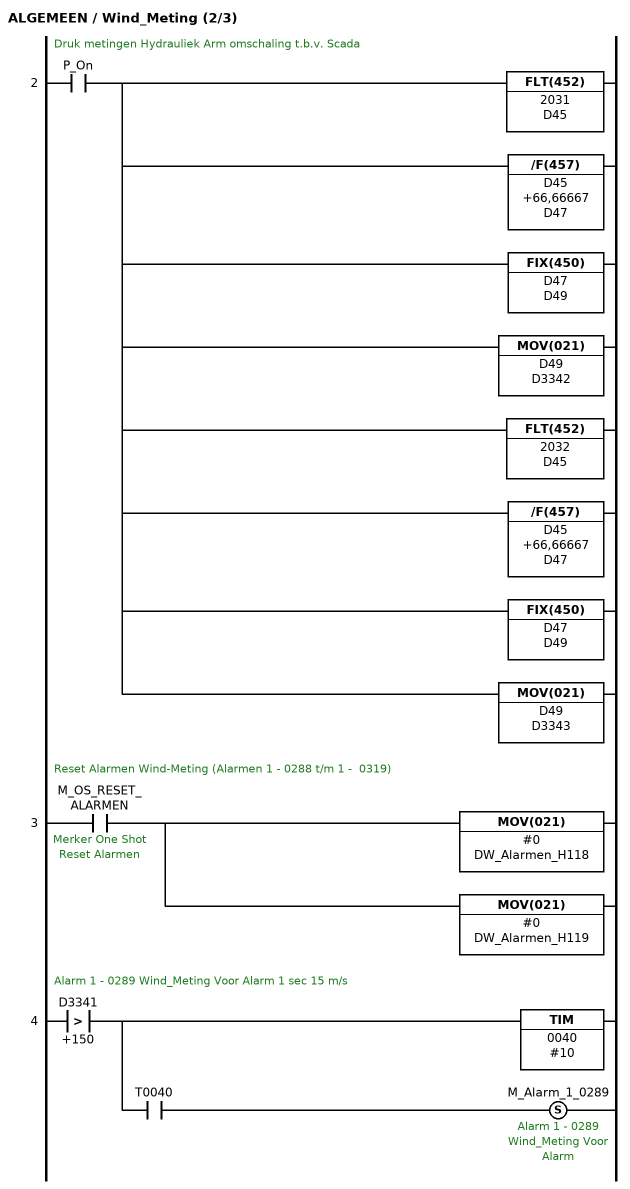
; rung 2: Druk metingen Hydrauliek Arm omschaling t.b.v. Scada
LD P_On
FLT(452) 2031 D45
/F(457) D45 +66,66667 D47
FIX(450) D47 D49
MOV(021) D49 D3342
FLT(452) 2032 D45
/F(457) D45 +66,66667 D47
FIX(450) D47 D49
MOV(021) D49 D3343
; rung 3: Reset Alarmen Wind-Meting (Alarmen 1 - 0288 t/m 1 -  0319)
LD M_OS_RESET_ALARMEN  ; Merker One Shot Reset Alarmen
MOV(021) #0 DW_Alarmen_H118
MOV(021) #0 DW_Alarmen_H119
; rung 4: Alarm 1 - 0289 Wind_Meting Voor Alarm 1 sec 15 m/s
LD>S(322) D3341 +150
TIM 0040 #10
AND T0040
SET M_Alarm_1_0289  ; Alarm 1 - 0289 Wind_Meting Voor Alarm

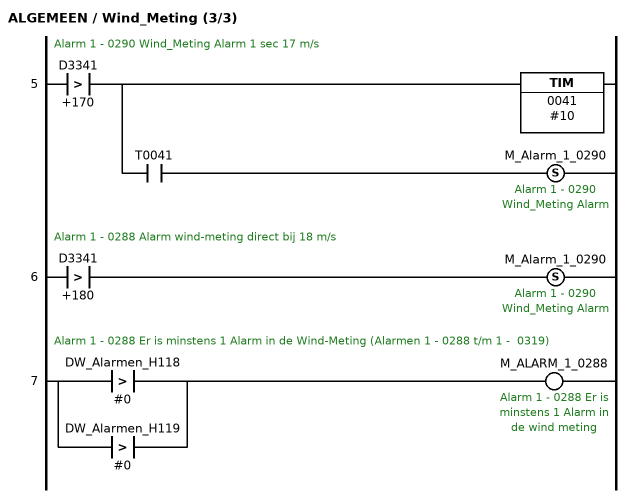
; rung 5: Alarm 1 - 0290 Wind_Meting Alarm 1 sec 17 m/s
LD>S(322) D3341 +170
TIM 0041 #10
AND T0041
SET M_Alarm_1_0290  ; Alarm 1 - 0290 Wind_Meting Alarm
; rung 6: Alarm 1 - 0288 Alarm wind-meting direct bij 18 m/s
LD>S(322) D3341 +180
SET M_Alarm_1_0290  ; Alarm 1 - 0290 Wind_Meting Alarm
; rung 7: Alarm 1 - 0288 Er is minstens 1 Alarm in de Wind-Meting (Alarmen 1 - 0288 t/m 1 -  0319)
LD>(320) DW_Alarmen_H118 #0
OR>(320) DW_Alarmen_H119 #0
OUT M_ALARM_1_0288  ; Alarm 1 - 0288 Er is minstens 1 Alarm in de wind meting

### Section Alarm_Handler

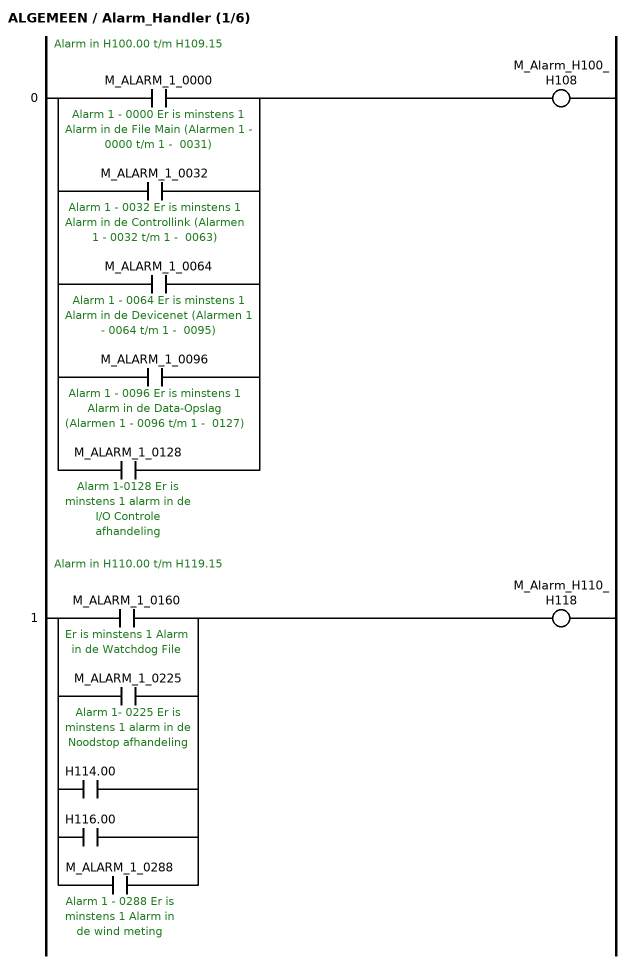
; rung 0: Alarm in H100.00 t/m H109.15
LD M_ALARM_1_0000  ; Alarm 1 - 0000 Er is minstens 1 Alarm in de File Main (Alarmen 1 - 0000 t/m 1 -  0031)
OR M_ALARM_1_0032  ; Alarm 1 - 0032 Er is minstens 1 Alarm in de Controllink (Alarmen 1 - 0032 t/m 1 -  0063)
OR M_ALARM_1_0064  ; Alarm 1 - 0064 Er is minstens 1 Alarm in de Devicenet (Alarmen 1 - 0064 t/m 1 -  0095)
OR M_ALARM_1_0096  ; Alarm 1 - 0096 Er is minstens 1 Alarm in de Data-Opslag (Alarmen 1 - 0096 t/m 1 -  0127)
OR M_ALARM_1_0128  ; Alarm 1-0128 Er is minstens 1 alarm in de I/O Controle afhandeling
OUT M_Alarm_H100_H108
; rung 1: Alarm in H110.00 t/m H119.15
LD M_ALARM_1_0160  ; Er is minstens 1 Alarm in de Watchdog File
OR M_ALARM_1_0225  ; Alarm 1- 0225 Er is minstens 1 alarm in de Noodstop afhandeling
OR H114.00
OR H116.00
OR M_ALARM_1_0288  ; Alarm 1 - 0288 Er is minstens 1 Alarm in de wind meting
OUT M_Alarm_H110_H118

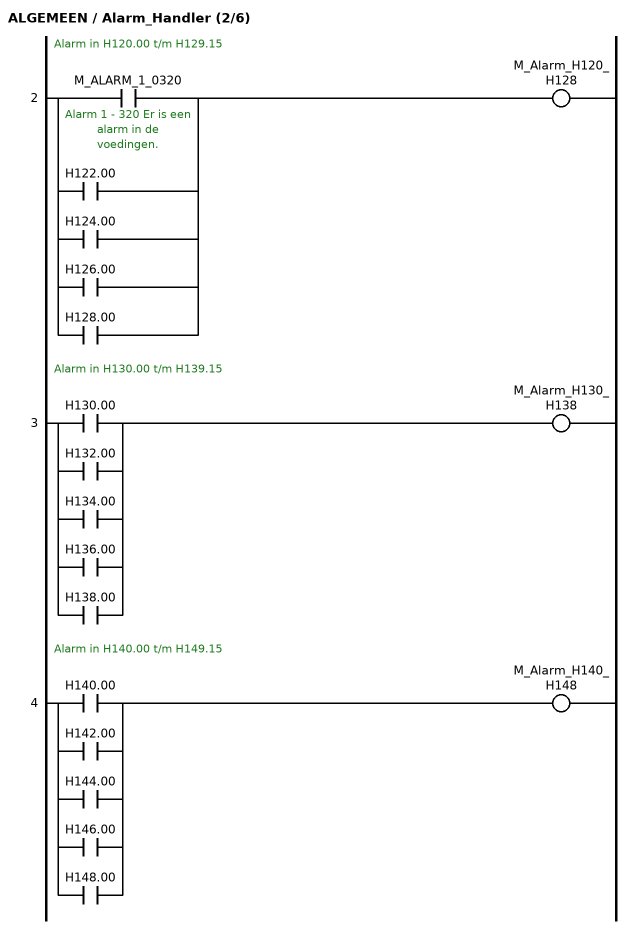
; rung 2: Alarm in H120.00 t/m H129.15
LD M_ALARM_1_0320  ; Alarm 1 - 320 Er is een alarm in de voedingen.
OR H122.00
OR H124.00
OR H126.00
OR H128.00
OUT M_Alarm_H120_H128
; rung 3: Alarm in H130.00 t/m H139.15
LD H130.00
OR H132.00
OR H134.00
OR H136.00
OR H138.00
OUT M_Alarm_H130_H138
; rung 4: Alarm in H140.00 t/m H149.15
LD H140.00
OR H142.00
OR H144.00
OR H146.00
OR H148.00
OUT M_Alarm_H140_H148

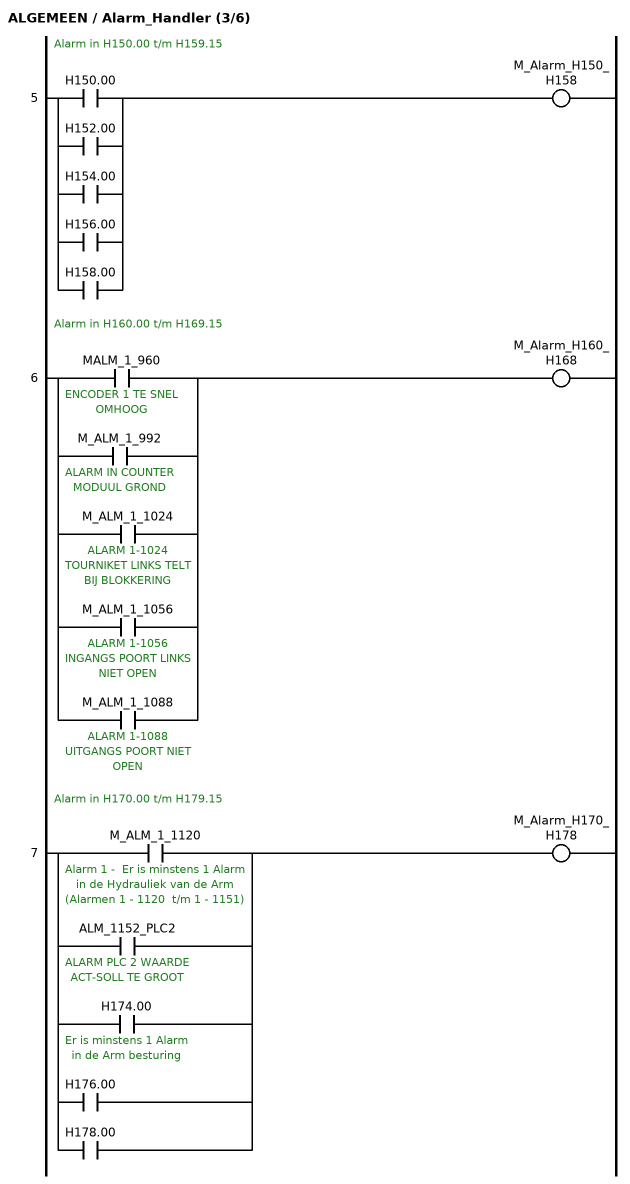
; rung 5: Alarm in H150.00 t/m H159.15
LD H150.00
OR H152.00
OR H154.00
OR H156.00
OR H158.00
OUT M_Alarm_H150_H158
; rung 6: Alarm in H160.00 t/m H169.15
LD MALM_1_960  ; ENCODER 1 TE SNEL OMHOOG
OR M_ALM_1_992  ; ALARM IN COUNTER MODUUL GROND
OR M_ALM_1_1024  ; ALARM 1-1024 TOURNIKET LINKS TELT BIJ BLOKKERING
OR M_ALM_1_1056  ; ALARM 1-1056 INGANGS POORT LINKS NIET OPEN
OR M_ALM_1_1088  ; ALARM 1-1088 UITGANGS POORT NIET OPEN
OUT M_Alarm_H160_H168
; rung 7: Alarm in H170.00 t/m H179.15
LD M_ALM_1_1120  ; Alarm 1 -  Er is minstens 1 Alarm in de Hydrauliek van de Arm  (Alarmen 1 - 1120  t/m 1 - 1151)
OR ALM_1152_PLC2  ; ALARM PLC 2 WAARDE ACT-SOLL TE GROOT
OR H174.00  ; Er is minstens 1 Alarm in de Arm besturing
OR H176.00
OR H178.00
OUT M_Alarm_H170_H178

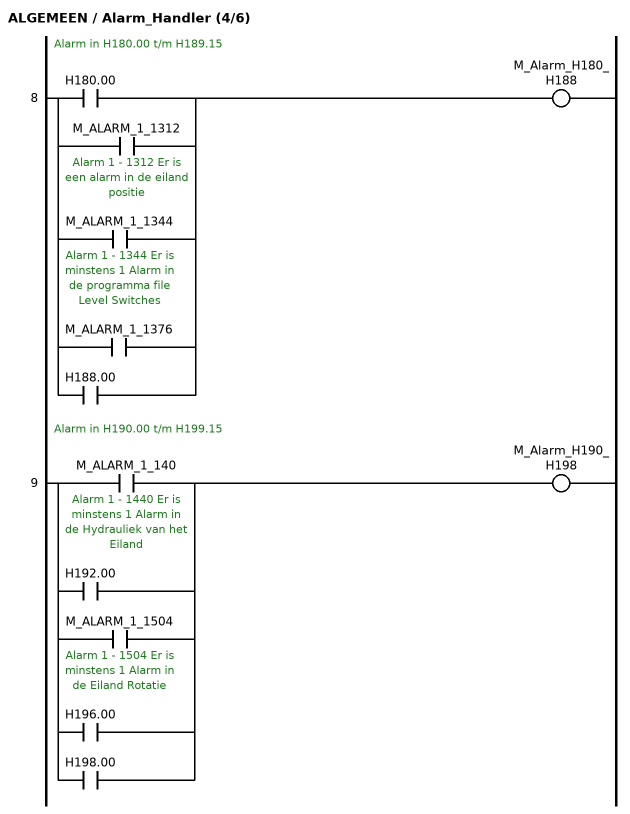
; rung 8: Alarm in H180.00 t/m H189.15
LD H180.00
OR M_ALARM_1_1312  ; Alarm 1 - 1312 Er is een alarm in de eiland positie
OR M_ALARM_1_1344  ; Alarm 1 - 1344 Er is minstens 1 Alarm in de programma file Level Switches
OR M_ALARM_1_1376
OR H188.00
OUT M_Alarm_H180_H188
; rung 9: Alarm in H190.00 t/m H199.15
LD M_ALARM_1_140  ; Alarm 1 - 1440 Er is minstens 1 Alarm in de Hydrauliek van het Eiland
OR H192.00
OR M_ALARM_1_1504  ; Alarm 1 - 1504 Er is minstens 1 Alarm in de Eiland Rotatie
OR H196.00
OR H198.00
OUT M_Alarm_H190_H198

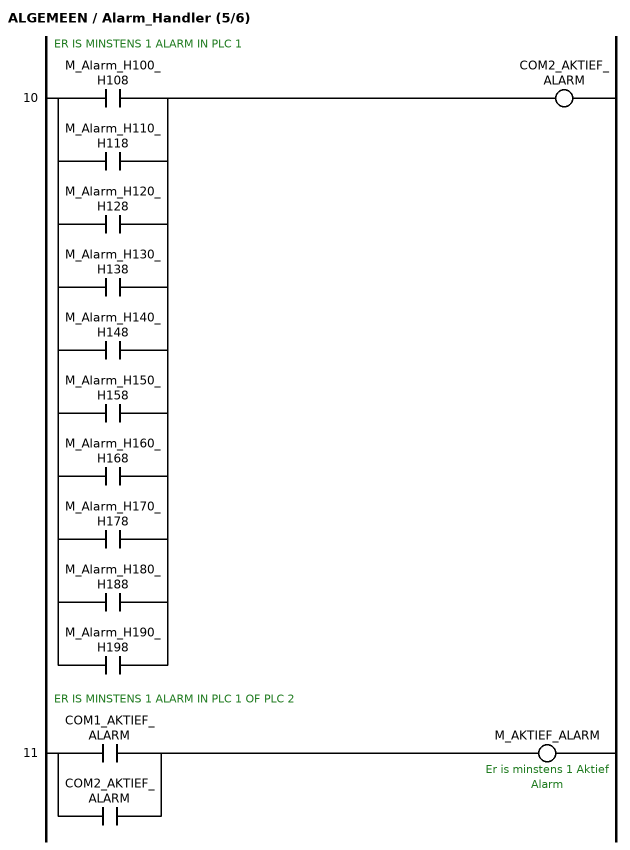
; rung 10: ER IS MINSTENS 1 ALARM IN PLC 1
LD M_Alarm_H100_H108
OR M_Alarm_H110_H118
OR M_Alarm_H120_H128
OR M_Alarm_H130_H138
OR M_Alarm_H140_H148
OR M_Alarm_H150_H158
OR M_Alarm_H160_H168
OR M_Alarm_H170_H178
OR M_Alarm_H180_H188
OR M_Alarm_H190_H198
OUT COM2_AKTIEF_ALARM
; rung 11: ER IS MINSTENS 1 ALARM IN PLC 1 OF PLC 2
LD COM1_AKTIEF_ALARM
OR COM2_AKTIEF_ALARM
OUT M_AKTIEF_ALARM  ; Er is minstens 1 Aktief Alarm

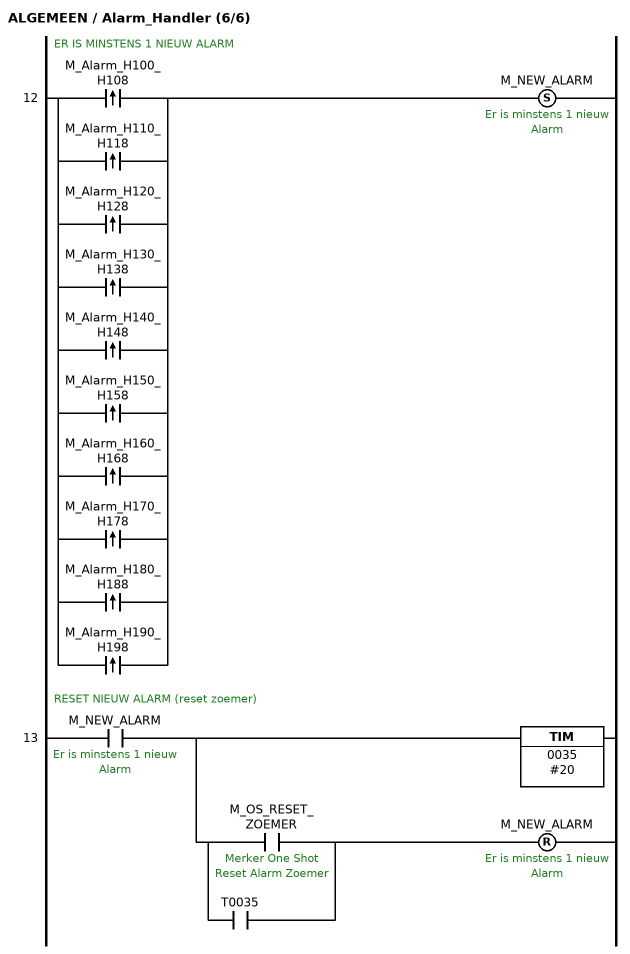
; rung 12: ER IS MINSTENS 1 NIEUW ALARM
@LD M_Alarm_H100_H108
@OR M_Alarm_H110_H118
@OR M_Alarm_H120_H128
@OR M_Alarm_H130_H138
@OR M_Alarm_H140_H148
@OR M_Alarm_H150_H158
@OR M_Alarm_H160_H168
@OR M_Alarm_H170_H178
@OR M_Alarm_H180_H188
@OR M_Alarm_H190_H198
SET M_NEW_ALARM  ; Er is minstens 1 nieuw Alarm
; rung 13: RESET NIEUW ALARM (reset zoemer)
LD M_NEW_ALARM  ; Er is minstens 1 nieuw Alarm
TIM 0035 #20
LD M_OS_RESET_ZOEMER  ; Merker One Shot Reset Alarm Zoemer
OR T0035
ANDLD
RSET M_NEW_ALARM  ; Er is minstens 1 nieuw Alarm

### Section Einde_Algemeen
; rung 0
END(001)

## Program BEDIENING_SIGNAAL (cyclic task 1)
Local symbols
Com1_44HS12 3011.15 BOOL
Com1_44HS124 3012.00 BOOL
Com1_SK_Open_Linker_Ingangs_Poortje_Eiland 3014.09 BOOL
Com1_SK_Open_Linker_Ingangs_Poortje_Oever 3014.11 BOOL
Com1_SK_Open_Linker_Uitgangs_Poortjes_Eiland 3014.13 BOOL
Com1_SK_Open_Rechter_Ingangs_Poortje_Eiland 3014.10 BOOL
Com1_SK_Open_Rechter_Ingangs_Poortje_Oever 3014.12 BOOL
Com1_SK_Open_Rechter_Uitgangs_Poortje_Eiland 3014.14 BOOL
Com1_SK_Open_Sluit_Linker_Oever_Poortjes_ 3014.05 BOOL
Com1_SK_Open_Sluit_Rechter_Oever_Poortjes_ 3014.06 BOOL
Com1_SK_Open_Uitgangs_Poortjes_Oever 3014.15 BOOL
Com1_SK_Reset_Alarmen 3014.01 BOOL
Com1_SK_SPARE_3314_00 3014.00 BOOL
Com1_SK_SPARE_3314_02 3014.02 BOOL
Com1_SK_SPARE_3315_03 3015.02 BOOL
Com1_SK_SPARE_3315_07 3015.07 BOOL
Com1_SK_SPARE_3315_08 3015.08 BOOL
Com1_SK_SPARE_3315_09 3015.09 BOOL
Com1_SK_Stabilisatie_Eiland_Linksom 3015.05 BOOL
Com1_SK_Stabilisatie_Eiland_Rechtsom 3015.06 BOOL
Com1_SK_Start_Stop_Hoofdpomp_Arm 3015.01 BOOL
Com1_SK_Start_Stop_Hoofdpomp_Eiland 3015.04 BOOL
Com1_SK_Start_Stop_Hydrau 3014.03 BOOL
Com1_SK_Start_Stop_Show 3014.04 BOOL
Com1_SK_Start_Stop_Stuurpomp_Arm 3015.00 BOOL
Com1_SK_Start_Stop_Stuurpomp_Eiland 3015.03 BOOL
Com1_SK_Vrijgave_Linker_Tourniquet 3014.07 BOOL
Com1_SK_Vrijgave_Rechter_Tourniquet 3014.08 BOOL
Com1_SK_WCD_1 3015.10 BOOL
Com1_SK_WCD_2 3015.11 BOOL
Com1_SK_WCD_3 3015.12 BOOL
Com1_SK_WCD_4 3015.13 BOOL
Com1_SK_WCD_5 3015.14 BOOL
Com1_SK_WCD_6 3015.15 BOOL
Com2_44HS14 3312.00 BOOL
Com2_SK_Open_Linker_Ingangs_Poortje_Eiland 3314.09 BOOL  ; Skada Bediening Open Linker Ingangs Poortje Eiland
Com2_SK_Open_Linker_Ingangs_Poortje_Oever 3314.11 BOOL  ; Skada Bediening Open Linker Ingangs Poortje Oever
Com2_SK_Open_Linker_Uitgangs_Poortjes_Eiland 3314.13 BOOL  ; Skada Bediening Open Linker Uitgangs Poortje Eiland
Com2_SK_Open_Rechter_Ingangs_Poortje_Eiland 3314.10 BOOL  ; Skada Bediening Open Rechter ingangs poortje Eiland
Com2_SK_Open_Rechter_Ingangs_Poortje_Oever 3314.12 BOOL  ; Skada Bediening Open Rechter ingangs poortje Oever
Com2_SK_Open_Rechter_Uitgangs_Poortje_Eiland 3314.14 BOOL  ; Skada Bediening Open Rechter Uitgangs poortje Eiland
Com2_SK_Open_Sluit_Linker_Oever_Poortjes_ 3314.05 BOOL  ; Skada Bediening Open / Sluit Linker Oever Poortjes
Com2_SK_Open_Sluit_Rechter_Oever_Poortjes_ 3314.06 BOOL  ; Skada Bediening Open / Sluit Rechter Oever Poortjes
Com2_SK_Open_Uitgangs_Poortjes_Oever 3314.15 BOOL  ; Skada Bediening Open Uitgangs poortjes Oever
Com2_SK_Reset_Alarmen 3314.01 BOOL  ; Skada Bediening Reset Alarmen
Com2_SK_SPARE_3314_00 3314.00 BOOL
Com2_SK_SPARE_3314_02 3314.02 BOOL
Com2_SK_SPARE_3315_03 3315.02 BOOL
Com2_SK_SPARE_3315_07 3315.07 BOOL
Com2_SK_SPARE_3315_08 3315.08 BOOL
Com2_SK_SPARE_3315_09 3315.09 BOOL
Com2_SK_Stabilisatie_Eiland_Linksom 3315.05 BOOL  ; Skada Bediening Eiland Stabilisatie Linksom
Com2_SK_Stabilisatie_Eiland_Rechtsom 3315.06 BOOL  ; Skada Bediening Eiland Stabilisatie Rechtsom
Com2_SK_Start_Stop_Hoofdpomp_Arm 3315.01 BOOL  ; Skada Bediening Start / Stop Hydrauliek Hoofdpomp Arm
Com2_SK_Start_Stop_Hoofdpomp_Eiland 3315.04 BOOL  ; Skada Bediening Start / Stop Hydrauliek Hoofdpomp Eiland
Com2_SK_Start_Stop_Hydrau 3314.03 BOOL  ; Skada Bediening Start / Stop Hydrauliek Arm & Eiland
Com2_SK_Start_Stop_Show 3314.04 BOOL  ; Skada Bediening Start / Stop Show
Com2_SK_Start_Stop_Stuurpomp_Arm 3315.00 BOOL  ; Skada Bediening Start / Stop Hydrauliek Stuurpomp Arm
Com2_SK_Start_Stop_Stuurpomp_Eiland 3315.03 BOOL  ; Skada Bediening Start / Stop Hydrauliek Stuurpomp Eiland
Com2_SK_Vrijgave_Linker_Tourniquet 3314.07 BOOL  ; Skada bediening Vrijgave Linker Tourniquets
Com2_SK_Vrijgave_Rechter_Tourniquet 3314.08 BOOL  ; Skada Bediening Vrijgave Rechter Tourniquets
Com2_SK_WCD_1 3315.10 BOOL  ; Skada Bediening Wandcontactdoos 1
Com2_SK_WCD_2 3315.11 BOOL  ; Skada Bediening Wandcontactdoos 2
Com2_SK_WCD_3 3315.12 BOOL  ; Skada Bediening Wandcontactdoos 3
Com2_SK_WCD_4 3315.13 BOOL  ; Skada Bediening Wandcontactdoos 4
Com2_SK_WCD_5 3315.14 BOOL  ; Skada Bediening Wandcontactdoos 5
Com2_SK_WCD_6 3315.15 BOOL  ; Skada Bediening Wandcontactdoos 6
Delay_Timer_Lamp_Test 0055 NUMBER  ; Delay Timer t.b.v. de lampen test
M_Hydrauliek_x_tijd_aan W56.03 BOOL  ; Hydrauliek x tijd laten door lopen nadat mode is veranderd

### Section Bediening_Scada

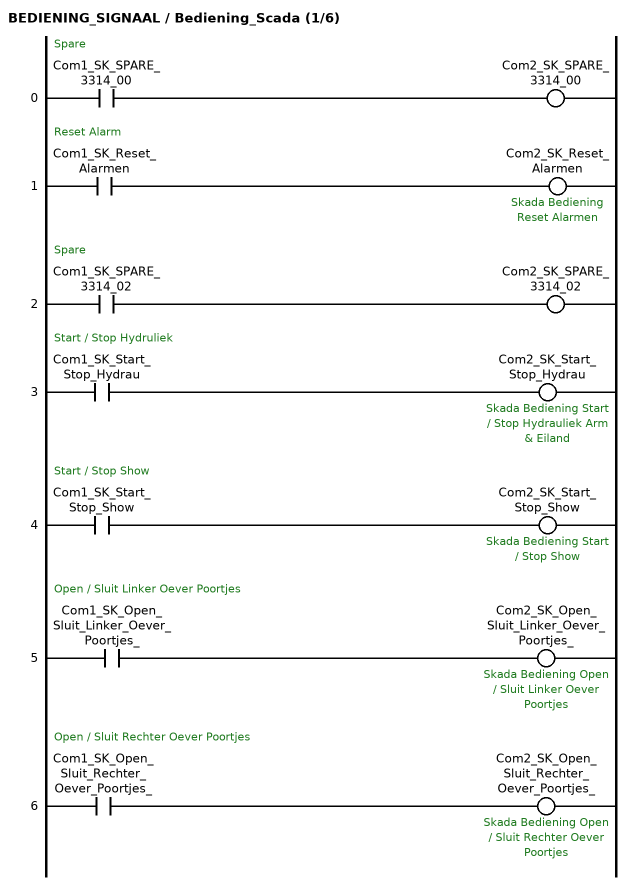
; rung 0: Spare
LD Com1_SK_SPARE_3314_00
OUT Com2_SK_SPARE_3314_00
; rung 1: Reset Alarm
LD Com1_SK_Reset_Alarmen
OUT Com2_SK_Reset_Alarmen  ; Skada Bediening Reset Alarmen
; rung 2: Spare
LD Com1_SK_SPARE_3314_02
OUT Com2_SK_SPARE_3314_02
; rung 3: Start / Stop Hydruliek
LD Com1_SK_Start_Stop_Hydrau
OUT Com2_SK_Start_Stop_Hydrau  ; Skada Bediening Start / Stop Hydrauliek Arm & Eiland
; rung 4: Start / Stop Show
LD Com1_SK_Start_Stop_Show
OUT Com2_SK_Start_Stop_Show  ; Skada Bediening Start / Stop Show
; rung 5: Open / Sluit Linker Oever Poortjes
LD Com1_SK_Open_Sluit_Linker_Oever_Poortjes_
OUT Com2_SK_Open_Sluit_Linker_Oever_Poortjes_  ; Skada Bediening Open / Sluit Linker Oever Poortjes
; rung 6: Open / Sluit Rechter Oever Poortjes
LD Com1_SK_Open_Sluit_Rechter_Oever_Poortjes_
OUT Com2_SK_Open_Sluit_Rechter_Oever_Poortjes_  ; Skada Bediening Open / Sluit Rechter Oever Poortjes

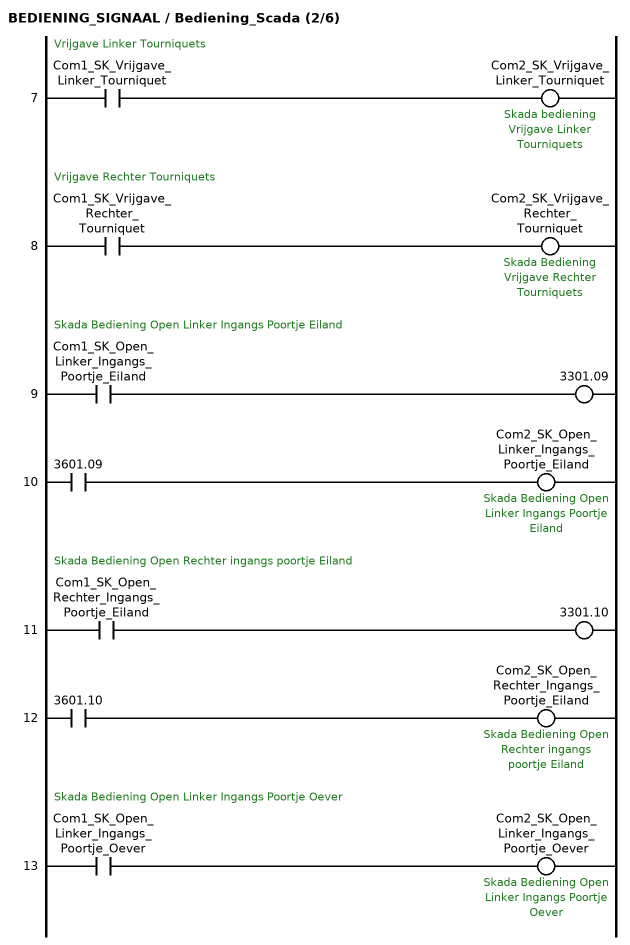
; rung 7: Vrijgave Linker Tourniquets
LD Com1_SK_Vrijgave_Linker_Tourniquet
OUT Com2_SK_Vrijgave_Linker_Tourniquet  ; Skada bediening Vrijgave Linker Tourniquets
; rung 8: Vrijgave Rechter Tourniquets
LD Com1_SK_Vrijgave_Rechter_Tourniquet
OUT Com2_SK_Vrijgave_Rechter_Tourniquet  ; Skada Bediening Vrijgave Rechter Tourniquets
; rung 9: Skada Bediening Open Linker Ingangs Poortje Eiland
LD Com1_SK_Open_Linker_Ingangs_Poortje_Eiland
OUT 3301.09
; rung 10
LD 3601.09
OUT Com2_SK_Open_Linker_Ingangs_Poortje_Eiland  ; Skada Bediening Open Linker Ingangs Poortje Eiland
; rung 11: Skada Bediening Open Rechter ingangs poortje Eiland
LD Com1_SK_Open_Rechter_Ingangs_Poortje_Eiland
OUT 3301.10
; rung 12
LD 3601.10
OUT Com2_SK_Open_Rechter_Ingangs_Poortje_Eiland  ; Skada Bediening Open Rechter ingangs poortje Eiland
; rung 13: Skada Bediening Open Linker Ingangs Poortje Oever
LD Com1_SK_Open_Linker_Ingangs_Poortje_Oever
OUT Com2_SK_Open_Linker_Ingangs_Poortje_Oever  ; Skada Bediening Open Linker Ingangs Poortje Oever

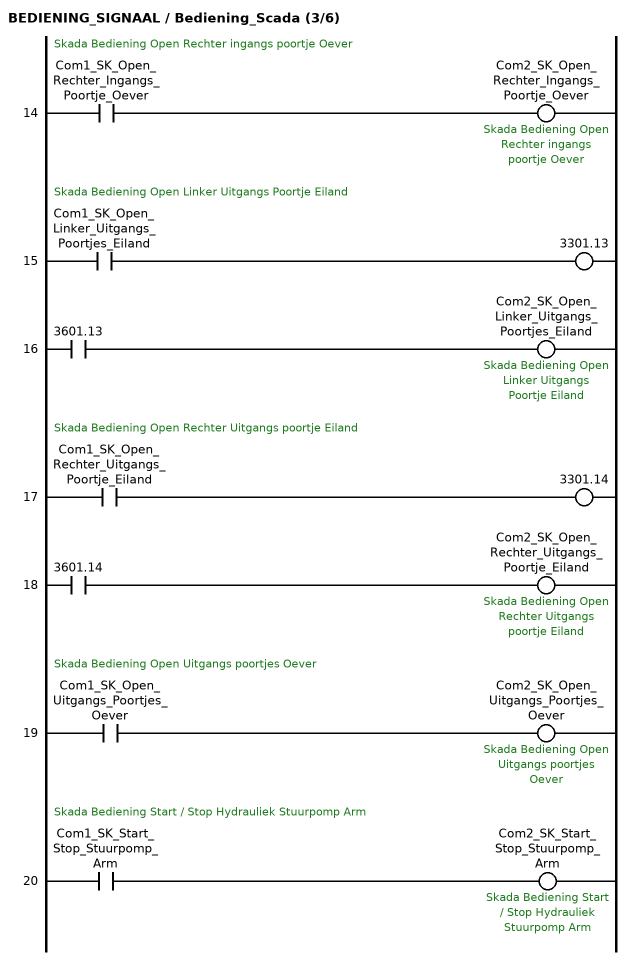
; rung 14: Skada Bediening Open Rechter ingangs poortje Oever
LD Com1_SK_Open_Rechter_Ingangs_Poortje_Oever
OUT Com2_SK_Open_Rechter_Ingangs_Poortje_Oever  ; Skada Bediening Open Rechter ingangs poortje Oever
; rung 15: Skada Bediening Open Linker Uitgangs Poortje Eiland
LD Com1_SK_Open_Linker_Uitgangs_Poortjes_Eiland
OUT 3301.13
; rung 16
LD 3601.13
OUT Com2_SK_Open_Linker_Uitgangs_Poortjes_Eiland  ; Skada Bediening Open Linker Uitgangs Poortje Eiland
; rung 17: Skada Bediening Open Rechter Uitgangs poortje Eiland
LD Com1_SK_Open_Rechter_Uitgangs_Poortje_Eiland
OUT 3301.14
; rung 18
LD 3601.14
OUT Com2_SK_Open_Rechter_Uitgangs_Poortje_Eiland  ; Skada Bediening Open Rechter Uitgangs poortje Eiland
; rung 19: Skada Bediening Open Uitgangs poortjes Oever
LD Com1_SK_Open_Uitgangs_Poortjes_Oever
OUT Com2_SK_Open_Uitgangs_Poortjes_Oever  ; Skada Bediening Open Uitgangs poortjes Oever
; rung 20: Skada Bediening Start / Stop Hydrauliek Stuurpomp Arm
LD Com1_SK_Start_Stop_Stuurpomp_Arm
OUT Com2_SK_Start_Stop_Stuurpomp_Arm  ; Skada Bediening Start / Stop Hydrauliek Stuurpomp Arm

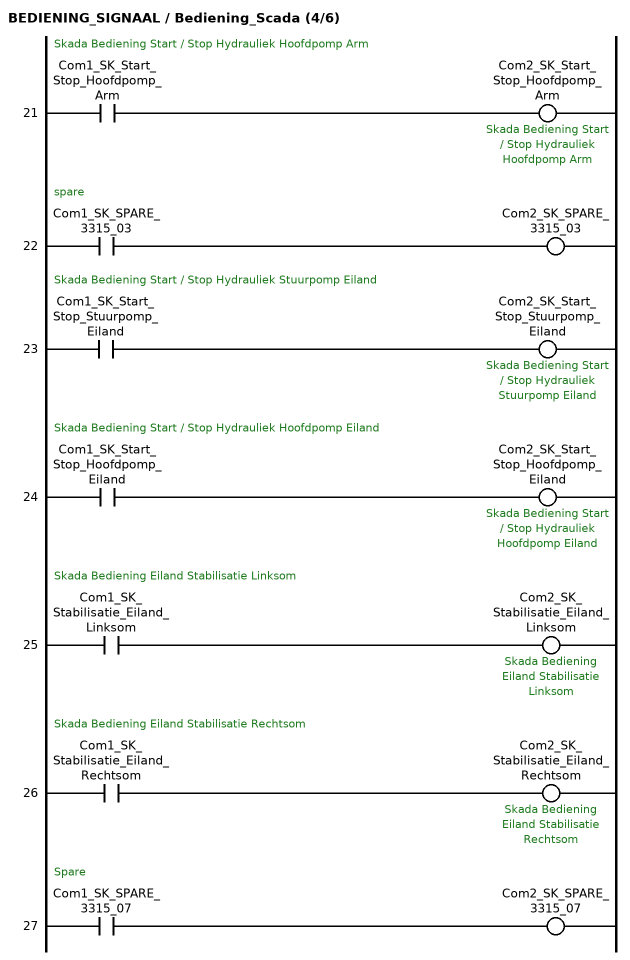
; rung 21: Skada Bediening Start / Stop Hydrauliek Hoofdpomp Arm
LD Com1_SK_Start_Stop_Hoofdpomp_Arm
OUT Com2_SK_Start_Stop_Hoofdpomp_Arm  ; Skada Bediening Start / Stop Hydrauliek Hoofdpomp Arm
; rung 22: spare
LD Com1_SK_SPARE_3315_03
OUT Com2_SK_SPARE_3315_03
; rung 23: Skada Bediening Start / Stop Hydrauliek Stuurpomp Eiland
LD Com1_SK_Start_Stop_Stuurpomp_Eiland
OUT Com2_SK_Start_Stop_Stuurpomp_Eiland  ; Skada Bediening Start / Stop Hydrauliek Stuurpomp Eiland
; rung 24: Skada Bediening Start / Stop Hydrauliek Hoofdpomp Eiland
LD Com1_SK_Start_Stop_Hoofdpomp_Eiland
OUT Com2_SK_Start_Stop_Hoofdpomp_Eiland  ; Skada Bediening Start / Stop Hydrauliek Hoofdpomp Eiland
; rung 25: Skada Bediening Eiland Stabilisatie Linksom
LD Com1_SK_Stabilisatie_Eiland_Linksom
OUT Com2_SK_Stabilisatie_Eiland_Linksom  ; Skada Bediening Eiland Stabilisatie Linksom
; rung 26: Skada Bediening Eiland Stabilisatie Rechtsom
LD Com1_SK_Stabilisatie_Eiland_Rechtsom
OUT Com2_SK_Stabilisatie_Eiland_Rechtsom  ; Skada Bediening Eiland Stabilisatie Rechtsom
; rung 27: Spare
LD Com1_SK_SPARE_3315_07
OUT Com2_SK_SPARE_3315_07

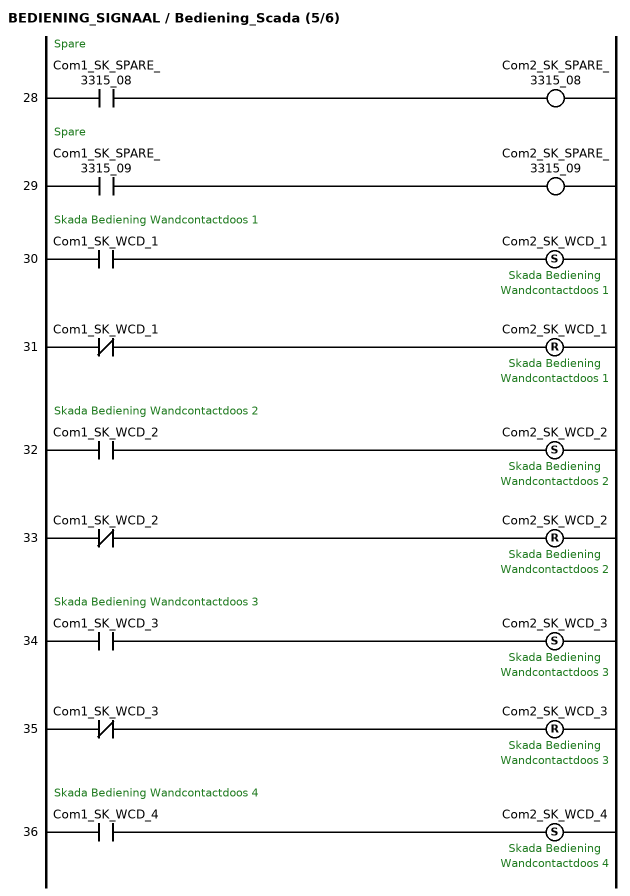
; rung 28: Spare
LD Com1_SK_SPARE_3315_08
OUT Com2_SK_SPARE_3315_08
; rung 29: Spare
LD Com1_SK_SPARE_3315_09
OUT Com2_SK_SPARE_3315_09
; rung 30: Skada Bediening Wandcontactdoos 1
LD Com1_SK_WCD_1
SET Com2_SK_WCD_1  ; Skada Bediening Wandcontactdoos 1
; rung 31
LDNOT Com1_SK_WCD_1
RSET Com2_SK_WCD_1  ; Skada Bediening Wandcontactdoos 1
; rung 32: Skada Bediening Wandcontactdoos 2
LD Com1_SK_WCD_2
SET Com2_SK_WCD_2  ; Skada Bediening Wandcontactdoos 2
; rung 33
LDNOT Com1_SK_WCD_2
RSET Com2_SK_WCD_2  ; Skada Bediening Wandcontactdoos 2
; rung 34: Skada Bediening Wandcontactdoos 3
LD Com1_SK_WCD_3
SET Com2_SK_WCD_3  ; Skada Bediening Wandcontactdoos 3
; rung 35
LDNOT Com1_SK_WCD_3
RSET Com2_SK_WCD_3  ; Skada Bediening Wandcontactdoos 3
; rung 36: Skada Bediening Wandcontactdoos 4
LD Com1_SK_WCD_4
SET Com2_SK_WCD_4  ; Skada Bediening Wandcontactdoos 4

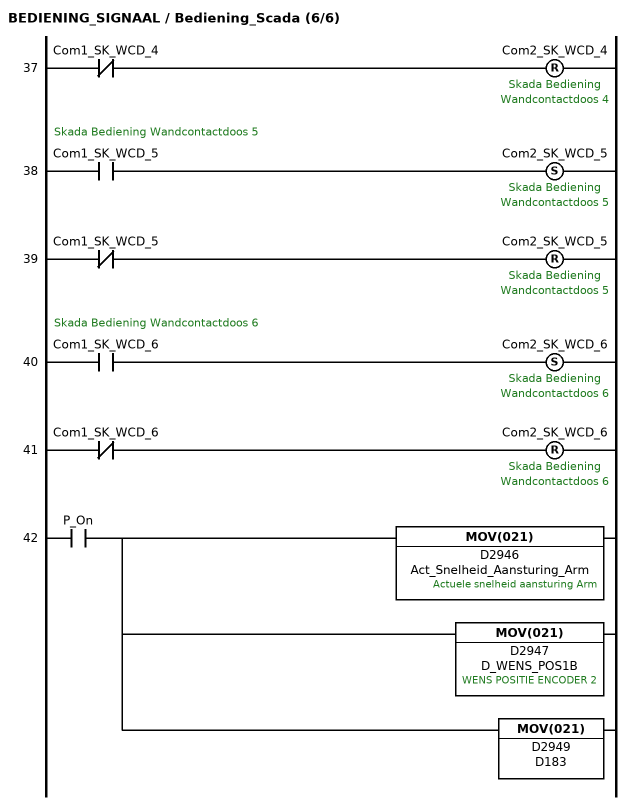
; rung 37
LDNOT Com1_SK_WCD_4
RSET Com2_SK_WCD_4  ; Skada Bediening Wandcontactdoos 4
; rung 38: Skada Bediening Wandcontactdoos 5
LD Com1_SK_WCD_5
SET Com2_SK_WCD_5  ; Skada Bediening Wandcontactdoos 5
; rung 39
LDNOT Com1_SK_WCD_5
RSET Com2_SK_WCD_5  ; Skada Bediening Wandcontactdoos 5
; rung 40: Skada Bediening Wandcontactdoos 6
LD Com1_SK_WCD_6
SET Com2_SK_WCD_6  ; Skada Bediening Wandcontactdoos 6
; rung 41
LDNOT Com1_SK_WCD_6
RSET Com2_SK_WCD_6  ; Skada Bediening Wandcontactdoos 6
; rung 42
LD P_On
MOV(021) D2946 Act_Snelheid_Aansturing_Arm  ; Actuele snelheid aansturing Arm
MOV(021) D2947 D_WENS_POS1B  ; WENS POSITIE ENCODER 2
MOV(021) D2949 D183

### Section Signalering_Scada

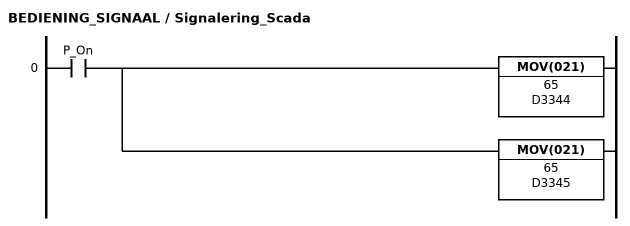
; rung 0
LD P_On
MOV(021) 65 D3344
MOV(021) 65 D3345

### Section Bediening_Grond

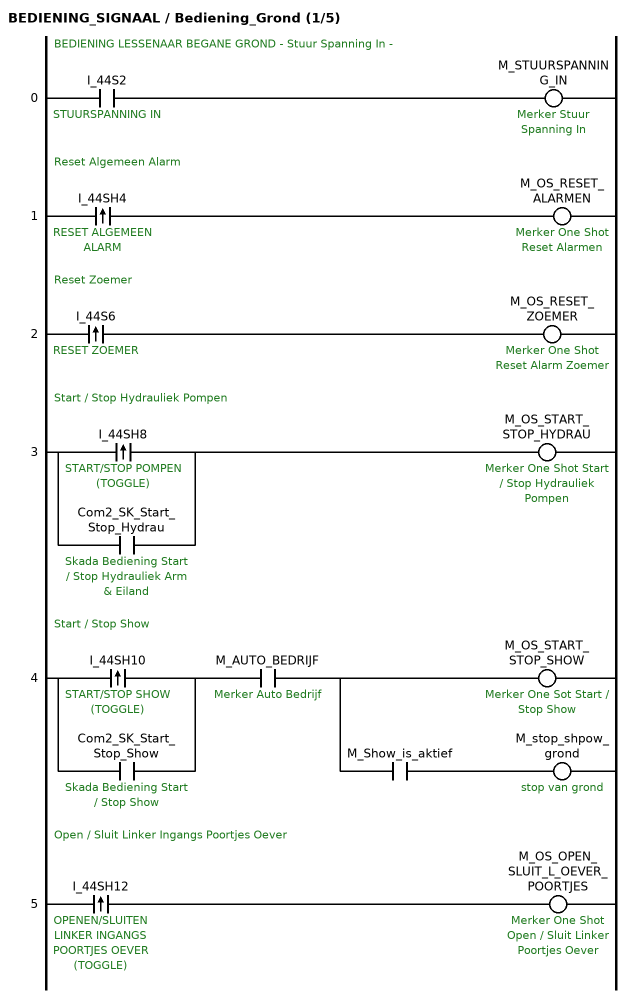
; rung 0: BEDIENING LESSENAAR BEGANE GROND - Stuur Spanning In -
LD I_44S2  ; STUURSPANNING IN
OUT M_STUURSPANNING_IN  ; Merker Stuur Spanning In
; rung 1: Reset Algemeen Alarm
@LD I_44SH4  ; RESET ALGEMEEN ALARM
OUT M_OS_RESET_ALARMEN  ; Merker One Shot Reset Alarmen
; rung 2: Reset Zoemer
@LD I_44S6  ; RESET ZOEMER
OUT M_OS_RESET_ZOEMER  ; Merker One Shot Reset Alarm Zoemer
; rung 3: Start / Stop Hydrauliek Pompen
@LD I_44SH8  ; START/STOP POMPEN (TOGGLE)
OR Com2_SK_Start_Stop_Hydrau  ; Skada Bediening Start / Stop Hydrauliek Arm & Eiland
OUT M_OS_START_STOP_HYDRAU  ; Merker One Shot Start / Stop Hydrauliek Pompen
; rung 4: Start / Stop Show
@LD I_44SH10  ; START/STOP SHOW (TOGGLE)
OR Com2_SK_Start_Stop_Show  ; Skada Bediening Start / Stop Show
AND M_AUTO_BEDRIJF  ; Merker Auto Bedrijf
OUT M_OS_START_STOP_SHOW  ; Merker One Sot Start / Stop Show
AND M_Show_is_aktief
OUT M_stop_shpow_grond  ; stop van grond
; rung 5: Open / Sluit Linker Ingangs Poortjes Oever
@LD I_44SH12  ; OPENEN/SLUITEN LINKER INGANGS POORTJES OEVER  (TOGGLE)
OUT M_OS_OPEN_SLUIT_L_OEVER_POORTJES  ; Merker One Shot Open / Sluit Linker Poortjes Oever

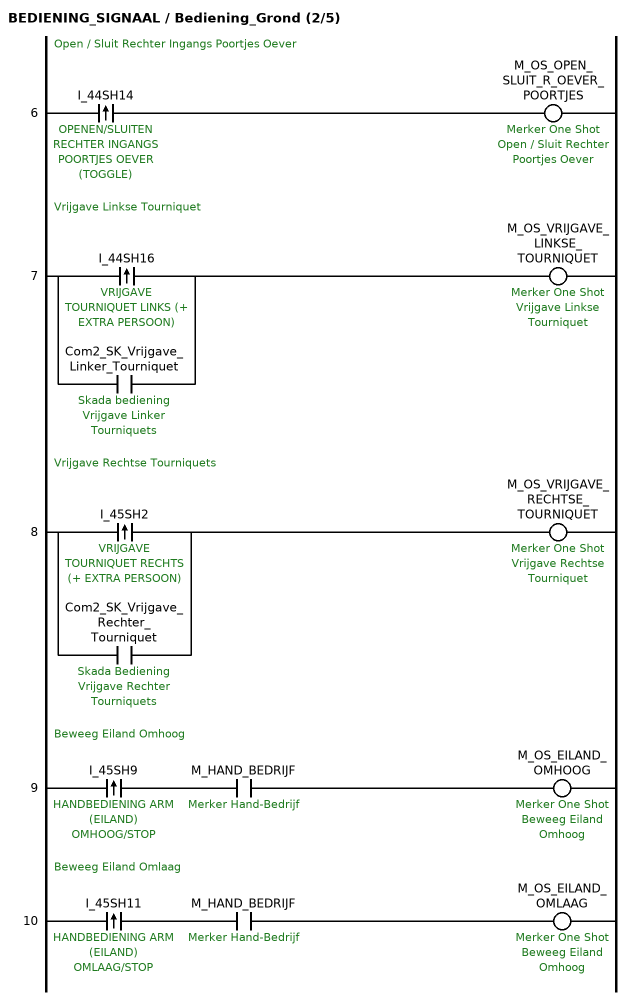
; rung 6: Open / Sluit Rechter Ingangs Poortjes Oever
@LD I_44SH14  ; OPENEN/SLUITEN RECHTER INGANGS POORTJES OEVER  (TOGGLE)
OUT M_OS_OPEN_SLUIT_R_OEVER_POORTJES  ; Merker One Shot Open / Sluit Rechter Poortjes Oever
; rung 7: Vrijgave Linkse Tourniquet
@LD I_44SH16  ; VRIJGAVE TOURNIQUET LINKS (+ EXTRA PERSOON)
OR Com2_SK_Vrijgave_Linker_Tourniquet  ; Skada bediening Vrijgave Linker Tourniquets
OUT M_OS_VRIJGAVE_LINKSE_TOURNIQUET  ; Merker One Shot Vrijgave Linkse Tourniquet
; rung 8: Vrijgave Rechtse Tourniquets
@LD I_45SH2  ; VRIJGAVE TOURNIQUET RECHTS (+ EXTRA PERSOON)
OR Com2_SK_Vrijgave_Rechter_Tourniquet  ; Skada Bediening Vrijgave Rechter Tourniquets
OUT M_OS_VRIJGAVE_RECHTSE_TOURNIQUET  ; Merker One Shot Vrijgave Rechtse Tourniquet
; rung 9: Beweeg Eiland Omhoog
@LD I_45SH9  ; HANDBEDIENING ARM (EILAND) OMHOOG/STOP
AND M_HAND_BEDRIJF  ; Merker Hand-Bedrijf
OUT M_OS_EILAND_OMHOOG  ; Merker One Shot Beweeg Eiland Omhoog
; rung 10: Beweeg Eiland Omlaag
@LD I_45SH11  ; HANDBEDIENING ARM (EILAND) OMLAAG/STOP
AND M_HAND_BEDRIJF  ; Merker Hand-Bedrijf
OUT M_OS_EILAND_OMLAAG  ; Merker One Shot Beweeg Eiland Omhoog

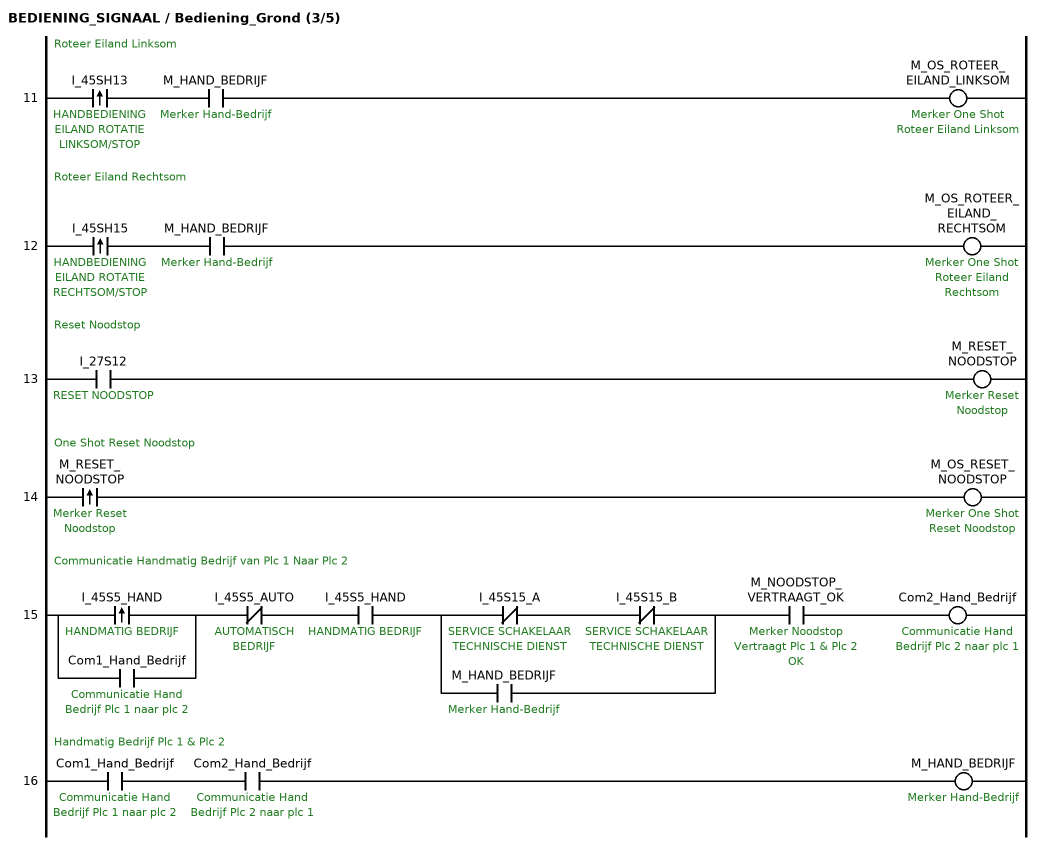
; rung 11: Roteer Eiland Linksom
@LD I_45SH13  ; HANDBEDIENING EILAND ROTATIE LINKSOM/STOP
AND M_HAND_BEDRIJF  ; Merker Hand-Bedrijf
OUT M_OS_ROTEER_EILAND_LINKSOM  ; Merker One Shot Roteer Eiland Linksom
; rung 12: Roteer Eiland Rechtsom
@LD I_45SH15  ; HANDBEDIENING EILAND ROTATIE RECHTSOM/STOP
AND M_HAND_BEDRIJF  ; Merker Hand-Bedrijf
OUT M_OS_ROTEER_EILAND_RECHTSOM  ; Merker One Shot Roteer Eiland Rechtsom
; rung 13: Reset Noodstop
LD I_27S12  ; RESET NOODSTOP
OUT M_RESET_NOODSTOP  ; Merker Reset Noodstop
; rung 14: One Shot Reset Noodstop
@LD M_RESET_NOODSTOP  ; Merker Reset Noodstop
OUT M_OS_RESET_NOODSTOP  ; Merker One Shot  Reset Noodstop
; rung 15: Communicatie Handmatig Bedrijf van Plc 1 Naar Plc 2
@LD I_45S5_HAND  ; HANDMATIG BEDRIJF
OR Com1_Hand_Bedrijf  ; Communicatie Hand Bedrijf Plc 1 naar plc 2
ANDNOT I_45S5_AUTO  ; AUTOMATISCH BEDRIJF
AND I_45S5_HAND  ; HANDMATIG BEDRIJF
LDNOT I_45S15_A  ; SERVICE SCHAKELAAR TECHNISCHE DIENST
ANDNOT I_45S15_B  ; SERVICE SCHAKELAAR TECHNISCHE DIENST
OR M_HAND_BEDRIJF  ; Merker Hand-Bedrijf
ANDLD
AND M_NOODSTOP_VERTRAAGT_OK  ; Merker Noodstop Vertraagt Plc 1 & Plc 2 OK
OUT Com2_Hand_Bedrijf  ; Communicatie Hand Bedrijf Plc 2 naar plc 1
; rung 16: Handmatig Bedrijf Plc 1 & Plc 2
LD Com1_Hand_Bedrijf  ; Communicatie Hand Bedrijf Plc 1 naar plc 2
AND Com2_Hand_Bedrijf  ; Communicatie Hand Bedrijf Plc 2 naar plc 1
OUT M_HAND_BEDRIJF  ; Merker Hand-Bedrijf

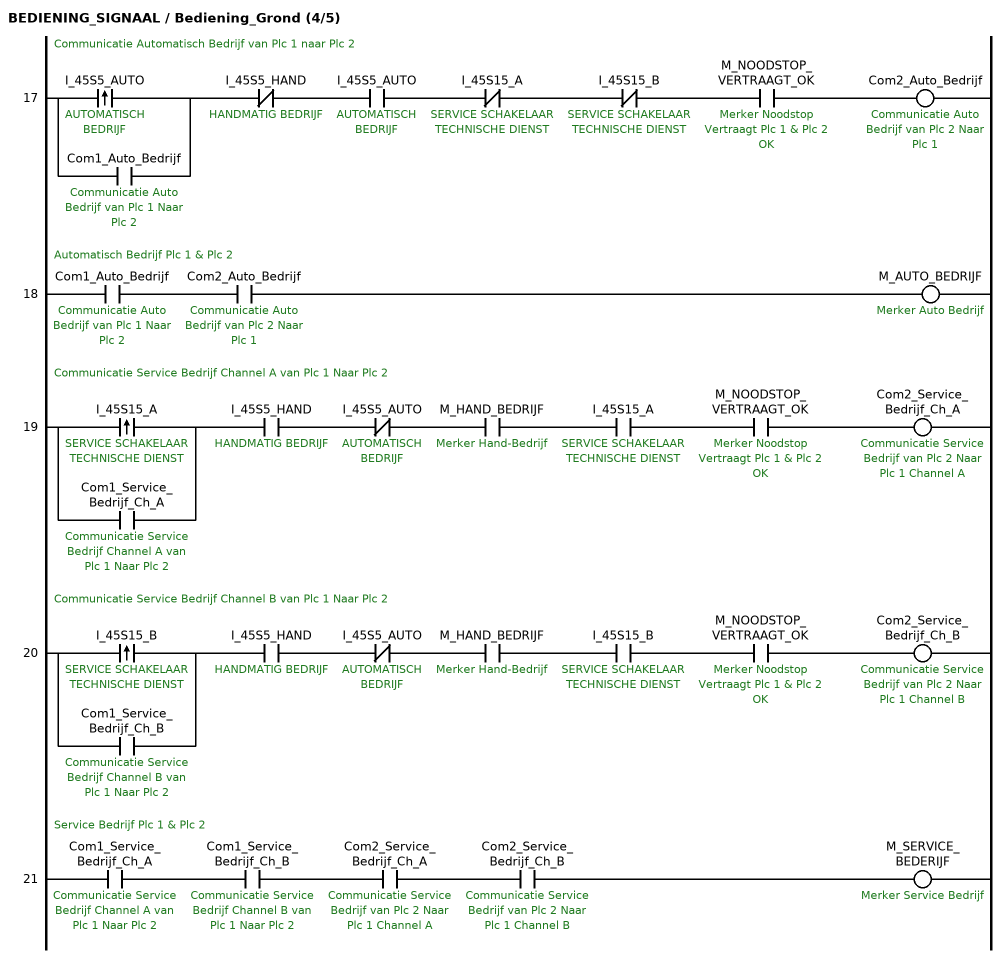
; rung 17: Communicatie Automatisch Bedrijf van Plc 1 naar Plc 2
@LD I_45S5_AUTO  ; AUTOMATISCH BEDRIJF
OR Com1_Auto_Bedrijf  ; Communicatie Auto Bedrijf van Plc 1 Naar Plc 2
ANDNOT I_45S5_HAND  ; HANDMATIG BEDRIJF
AND I_45S5_AUTO  ; AUTOMATISCH BEDRIJF
ANDNOT I_45S15_A  ; SERVICE SCHAKELAAR TECHNISCHE DIENST
ANDNOT I_45S15_B  ; SERVICE SCHAKELAAR TECHNISCHE DIENST
AND M_NOODSTOP_VERTRAAGT_OK  ; Merker Noodstop Vertraagt Plc 1 & Plc 2 OK
OUT Com2_Auto_Bedrijf  ; Communicatie Auto Bedrijf van Plc 2 Naar Plc 1
; rung 18: Automatisch Bedrijf Plc 1 & Plc 2
LD Com1_Auto_Bedrijf  ; Communicatie Auto Bedrijf van Plc 1 Naar Plc 2
AND Com2_Auto_Bedrijf  ; Communicatie Auto Bedrijf van Plc 2 Naar Plc 1
OUT M_AUTO_BEDRIJF  ; Merker Auto Bedrijf
; rung 19: Communicatie Service Bedrijf Channel A van Plc 1 Naar Plc 2
@LD I_45S15_A  ; SERVICE SCHAKELAAR TECHNISCHE DIENST
OR Com1_Service_Bedrijf_Ch_A  ; Communicatie Service Bedrijf Channel A van Plc 1 Naar Plc 2
AND I_45S5_HAND  ; HANDMATIG BEDRIJF
ANDNOT I_45S5_AUTO  ; AUTOMATISCH BEDRIJF
AND M_HAND_BEDRIJF  ; Merker Hand-Bedrijf
AND I_45S15_A  ; SERVICE SCHAKELAAR TECHNISCHE DIENST
AND M_NOODSTOP_VERTRAAGT_OK  ; Merker Noodstop Vertraagt Plc 1 & Plc 2 OK
OUT Com2_Service_Bedrijf_Ch_A  ; Communicatie Service Bedrijf van Plc 2 Naar Plc 1 Channel A
; rung 20: Communicatie Service Bedrijf Channel B van Plc 1 Naar Plc 2
@LD I_45S15_B  ; SERVICE SCHAKELAAR TECHNISCHE DIENST
OR Com1_Service_Bedrijf_Ch_B  ; Communicatie Service Bedrijf Channel B van Plc 1 Naar Plc 2
AND I_45S5_HAND  ; HANDMATIG BEDRIJF
ANDNOT I_45S5_AUTO  ; AUTOMATISCH BEDRIJF
AND M_HAND_BEDRIJF  ; Merker Hand-Bedrijf
AND I_45S15_B  ; SERVICE SCHAKELAAR TECHNISCHE DIENST
AND M_NOODSTOP_VERTRAAGT_OK  ; Merker Noodstop Vertraagt Plc 1 & Plc 2 OK
OUT Com2_Service_Bedrijf_Ch_B  ; Communicatie Service Bedrijf van Plc 2 Naar Plc 1 Channel B
; rung 21: Service Bedrijf Plc 1 & Plc 2
LD Com1_Service_Bedrijf_Ch_A  ; Communicatie Service Bedrijf Channel A van Plc 1 Naar Plc 2
AND Com1_Service_Bedrijf_Ch_B  ; Communicatie Service Bedrijf Channel B van Plc 1 Naar Plc 2
AND Com2_Service_Bedrijf_Ch_A  ; Communicatie Service Bedrijf van Plc 2 Naar Plc 1 Channel A
AND Com2_Service_Bedrijf_Ch_B  ; Communicatie Service Bedrijf van Plc 2 Naar Plc 1 Channel B
OUT M_SERVICE_BEDERIJF  ; Merker Service Bedrijf

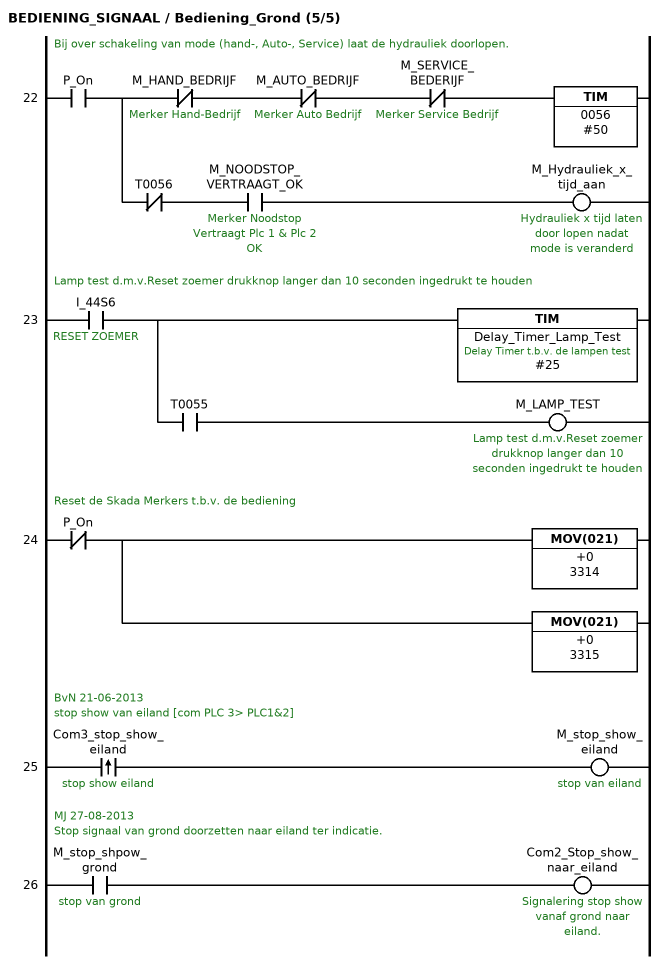
; rung 22: Bij over schakeling van mode (hand-, Auto-, Service) laat de hydrauliek doorlopen.
LD P_On
OUT TR0
ANDNOT M_HAND_BEDRIJF  ; Merker Hand-Bedrijf
ANDNOT M_AUTO_BEDRIJF  ; Merker Auto Bedrijf
ANDNOT M_SERVICE_BEDERIJF  ; Merker Service Bedrijf
TIM 0056 #50
LD TR0
ANDNOT T0056
AND M_NOODSTOP_VERTRAAGT_OK  ; Merker Noodstop Vertraagt Plc 1 & Plc 2 OK
OUT M_Hydrauliek_x_tijd_aan  ; Hydrauliek x tijd laten door lopen nadat mode is veranderd
; rung 23: Lamp test d.m.v.Reset zoemer drukknop langer dan 10 seconden ingedrukt te houden
LD I_44S6  ; RESET ZOEMER
TIM Delay_Timer_Lamp_Test #25  ; Delay Timer t.b.v. de lampen test
AND T0055
OUT M_LAMP_TEST  ; Lamp test d.m.v.Reset zoemer drukknop langer dan 10 seconden ingedrukt te houden
; rung 24: Reset de Skada Merkers t.b.v. de bediening
LDNOT P_On
MOV(021) +0 3314
MOV(021) +0 3315
; rung 25: BvN 21-06-2013 / stop show van eiland [com PLC 3> PLC1&2]
@LD Com3_stop_show_eiland  ; stop show eiland
OUT M_stop_show_eiland  ; stop van eiland
; rung 26: MJ 27-08-2013 / Stop signaal van grond doorzetten naar eiland ter indicatie.
LD M_stop_shpow_grond  ; stop van grond
OUT Com2_Stop_show_naar_eiland  ; Signalering stop show vanaf grond naar eiland.

### Section Signalering_Grond

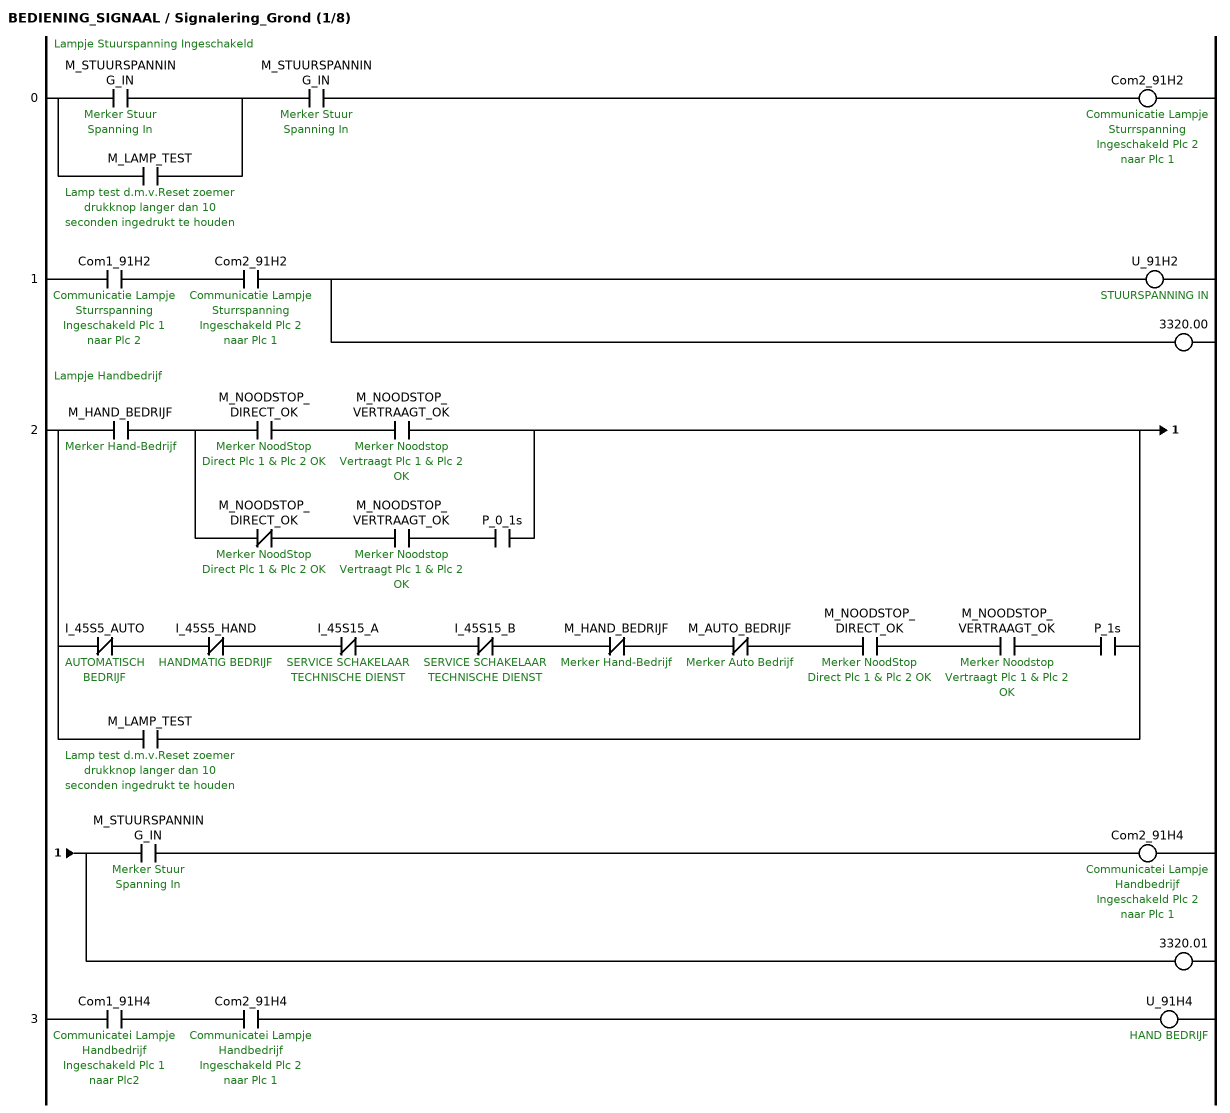
; rung 0: Lampje Stuurspanning Ingeschakeld
LD M_STUURSPANNING_IN  ; Merker Stuur Spanning In
OR M_LAMP_TEST  ; Lamp test d.m.v.Reset zoemer drukknop langer dan 10 seconden ingedrukt te houden
AND M_STUURSPANNING_IN  ; Merker Stuur Spanning In
OUT Com2_91H2  ; Communicatie Lampje Sturrspanning Ingeschakeld Plc 2 naar Plc 1
; rung 1
LD Com1_91H2  ; Communicatie Lampje Sturrspanning Ingeschakeld Plc 1 naar Plc 2
AND Com2_91H2  ; Communicatie Lampje Sturrspanning Ingeschakeld Plc 2 naar Plc 1
OUT U_91H2  ; STUURSPANNING IN
OUT 3320.00
; rung 2: Lampje Handbedrijf
LD M_HAND_BEDRIJF  ; Merker Hand-Bedrijf
LD M_NOODSTOP_DIRECT_OK  ; Merker NoodStop Direct Plc 1 & Plc 2 OK
AND M_NOODSTOP_VERTRAAGT_OK  ; Merker Noodstop Vertraagt Plc 1 & Plc 2 OK
LDNOT M_NOODSTOP_DIRECT_OK  ; Merker NoodStop Direct Plc 1 & Plc 2 OK
AND M_NOODSTOP_VERTRAAGT_OK  ; Merker Noodstop Vertraagt Plc 1 & Plc 2 OK
AND P_0_1s
ORLD
ANDLD
LDNOT I_45S5_AUTO  ; AUTOMATISCH BEDRIJF
ANDNOT I_45S5_HAND  ; HANDMATIG BEDRIJF
ANDNOT I_45S15_A  ; SERVICE SCHAKELAAR TECHNISCHE DIENST
ANDNOT I_45S15_B  ; SERVICE SCHAKELAAR TECHNISCHE DIENST
ANDNOT M_HAND_BEDRIJF  ; Merker Hand-Bedrijf
ANDNOT M_AUTO_BEDRIJF  ; Merker Auto Bedrijf
AND M_NOODSTOP_DIRECT_OK  ; Merker NoodStop Direct Plc 1 & Plc 2 OK
AND M_NOODSTOP_VERTRAAGT_OK  ; Merker Noodstop Vertraagt Plc 1 & Plc 2 OK
AND P_1s
ORLD
OR M_LAMP_TEST  ; Lamp test d.m.v.Reset zoemer drukknop langer dan 10 seconden ingedrukt te houden
OUT TR0
AND M_STUURSPANNING_IN  ; Merker Stuur Spanning In
OUT Com2_91H4  ; Communicatei Lampje Handbedrijf Ingeschakeld Plc 2 naar Plc 1
LD TR0
OUT 3320.01
; rung 3
LD Com1_91H4  ; Communicatei Lampje Handbedrijf Ingeschakeld Plc 1 naar Plc2
AND Com2_91H4  ; Communicatei Lampje Handbedrijf Ingeschakeld Plc 2 naar Plc 1
OUT U_91H4  ; HAND BEDRIJF

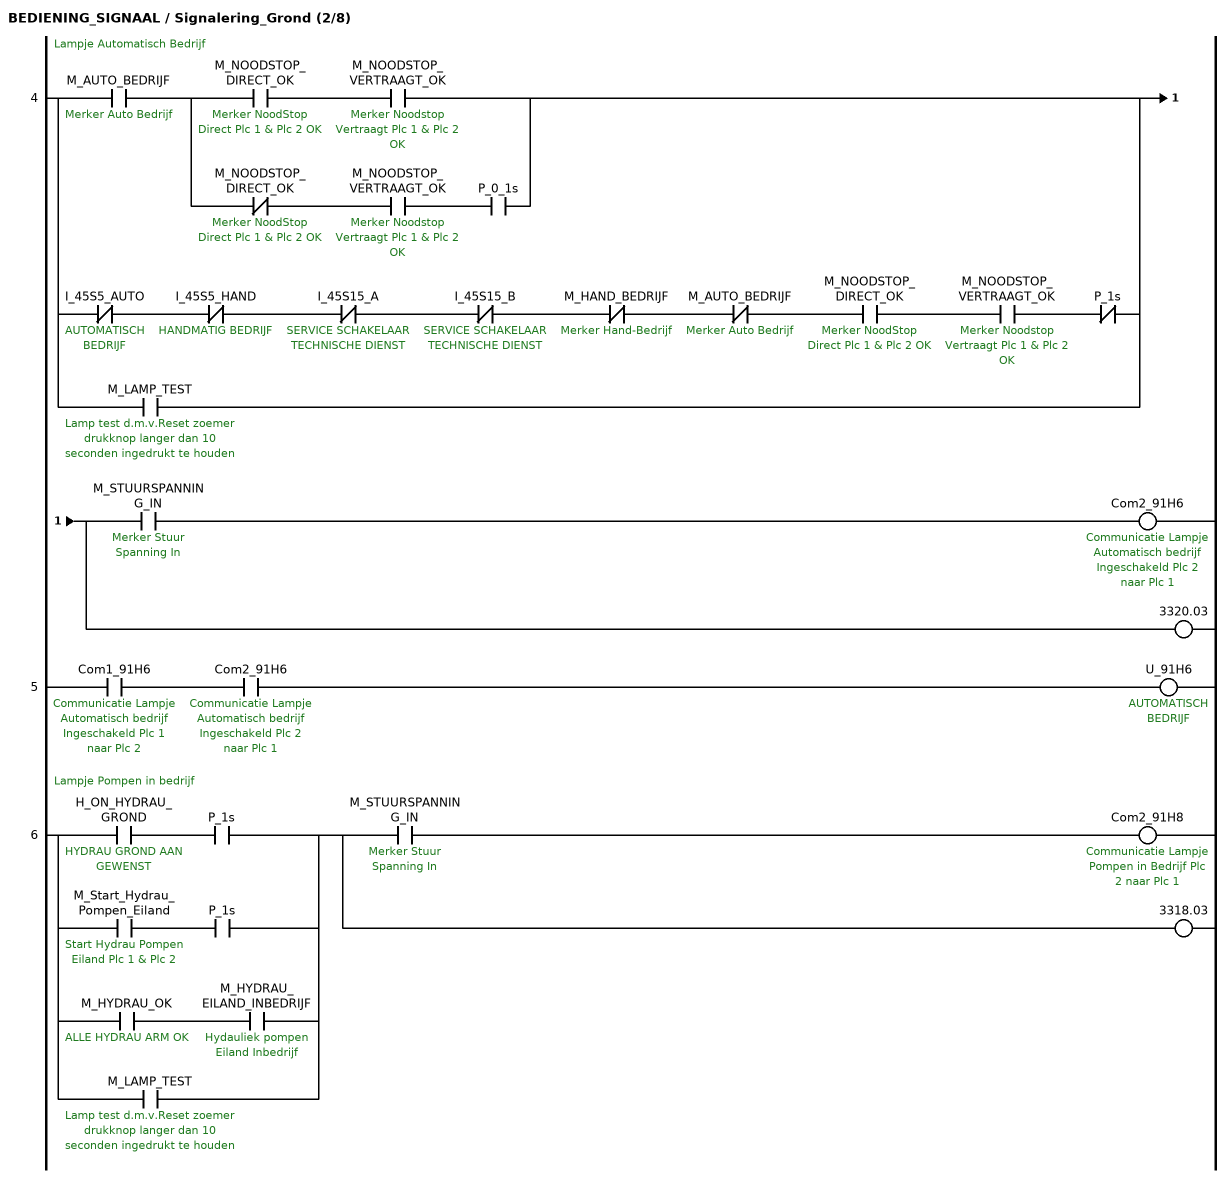
; rung 4: Lampje Automatisch Bedrijf
LD M_AUTO_BEDRIJF  ; Merker Auto Bedrijf
LD M_NOODSTOP_DIRECT_OK  ; Merker NoodStop Direct Plc 1 & Plc 2 OK
AND M_NOODSTOP_VERTRAAGT_OK  ; Merker Noodstop Vertraagt Plc 1 & Plc 2 OK
LDNOT M_NOODSTOP_DIRECT_OK  ; Merker NoodStop Direct Plc 1 & Plc 2 OK
AND M_NOODSTOP_VERTRAAGT_OK  ; Merker Noodstop Vertraagt Plc 1 & Plc 2 OK
AND P_0_1s
ORLD
ANDLD
LDNOT I_45S5_AUTO  ; AUTOMATISCH BEDRIJF
ANDNOT I_45S5_HAND  ; HANDMATIG BEDRIJF
ANDNOT I_45S15_A  ; SERVICE SCHAKELAAR TECHNISCHE DIENST
ANDNOT I_45S15_B  ; SERVICE SCHAKELAAR TECHNISCHE DIENST
ANDNOT M_HAND_BEDRIJF  ; Merker Hand-Bedrijf
ANDNOT M_AUTO_BEDRIJF  ; Merker Auto Bedrijf
AND M_NOODSTOP_DIRECT_OK  ; Merker NoodStop Direct Plc 1 & Plc 2 OK
AND M_NOODSTOP_VERTRAAGT_OK  ; Merker Noodstop Vertraagt Plc 1 & Plc 2 OK
ANDNOT P_1s
ORLD
OR M_LAMP_TEST  ; Lamp test d.m.v.Reset zoemer drukknop langer dan 10 seconden ingedrukt te houden
OUT TR0
AND M_STUURSPANNING_IN  ; Merker Stuur Spanning In
OUT Com2_91H6  ; Communicatie Lampje Automatisch bedrijf Ingeschakeld Plc 2 naar Plc 1
LD TR0
OUT 3320.03
; rung 5
LD Com1_91H6  ; Communicatie Lampje Automatisch bedrijf Ingeschakeld Plc 1 naar Plc 2
AND Com2_91H6  ; Communicatie Lampje Automatisch bedrijf Ingeschakeld Plc 2 naar Plc 1
OUT U_91H6  ; AUTOMATISCH BEDRIJF
; rung 6: Lampje Pompen in bedrijf
LD H_ON_HYDRAU_GROND  ; HYDRAU GROND AAN GEWENST
AND P_1s
LD M_Start_Hydrau_Pompen_Eiland  ; Start Hydrau Pompen Eiland Plc 1 & Plc 2
AND P_1s
ORLD
LD M_HYDRAU_OK  ; ALLE HYDRAU ARM OK
AND M_HYDRAU_EILAND_INBEDRIJF  ; Hydauliek pompen Eiland Inbedrijf
ORLD
OR M_LAMP_TEST  ; Lamp test d.m.v.Reset zoemer drukknop langer dan 10 seconden ingedrukt te houden
OUT TR0
AND M_STUURSPANNING_IN  ; Merker Stuur Spanning In
OUT Com2_91H8  ; Communicatie Lampje Pompen in Bedrijf Plc 2 naar Plc 1
LD TR0
OUT 3318.03

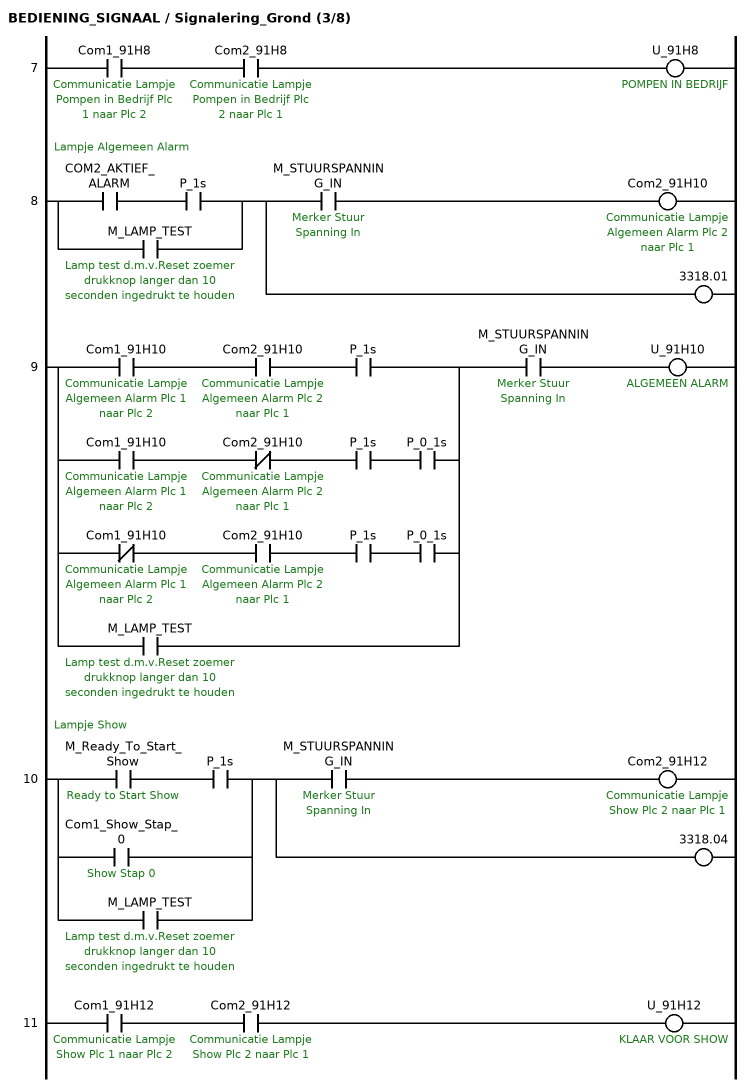
; rung 7
LD Com1_91H8  ; Communicatie Lampje Pompen in Bedrijf Plc 1 naar Plc 2
AND Com2_91H8  ; Communicatie Lampje Pompen in Bedrijf Plc 2 naar Plc 1
OUT U_91H8  ; POMPEN IN BEDRIJF
; rung 8: Lampje Algemeen Alarm
LD COM2_AKTIEF_ALARM
AND P_1s
OR M_LAMP_TEST  ; Lamp test d.m.v.Reset zoemer drukknop langer dan 10 seconden ingedrukt te houden
OUT TR0
AND M_STUURSPANNING_IN  ; Merker Stuur Spanning In
OUT Com2_91H10  ; Communicatie Lampje Algemeen Alarm Plc 2 naar Plc 1
LD TR0
OUT 3318.01
; rung 9
LD Com1_91H10  ; Communicatie Lampje Algemeen Alarm Plc 1 naar Plc 2
AND Com2_91H10  ; Communicatie Lampje Algemeen Alarm Plc 2 naar Plc 1
AND P_1s
LD Com1_91H10  ; Communicatie Lampje Algemeen Alarm Plc 1 naar Plc 2
ANDNOT Com2_91H10  ; Communicatie Lampje Algemeen Alarm Plc 2 naar Plc 1
AND P_1s
AND P_0_1s
ORLD
LDNOT Com1_91H10  ; Communicatie Lampje Algemeen Alarm Plc 1 naar Plc 2
AND Com2_91H10  ; Communicatie Lampje Algemeen Alarm Plc 2 naar Plc 1
AND P_1s
AND P_0_1s
ORLD
OR M_LAMP_TEST  ; Lamp test d.m.v.Reset zoemer drukknop langer dan 10 seconden ingedrukt te houden
AND M_STUURSPANNING_IN  ; Merker Stuur Spanning In
OUT U_91H10  ; ALGEMEEN ALARM
; rung 10: Lampje Show
LD M_Ready_To_Start_Show  ; Ready to Start Show
AND P_1s
OR Com1_Show_Stap_0  ; Show Stap 0
OR M_LAMP_TEST  ; Lamp test d.m.v.Reset zoemer drukknop langer dan 10 seconden ingedrukt te houden
OUT TR0
AND M_STUURSPANNING_IN  ; Merker Stuur Spanning In
OUT Com2_91H12  ; Communicatie Lampje Show Plc 2 naar Plc 1
LD TR0
OUT 3318.04
; rung 11
LD Com1_91H12  ; Communicatie Lampje Show Plc 1 naar Plc 2
AND Com2_91H12  ; Communicatie Lampje Show Plc 2 naar Plc 1
OUT U_91H12  ; KLAAR VOOR SHOW

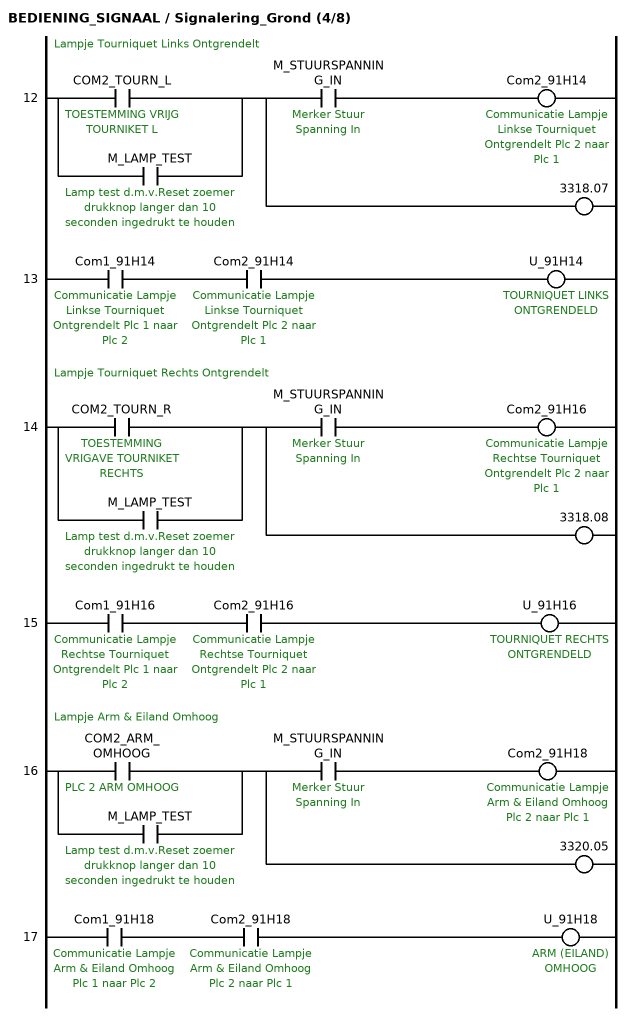
; rung 12: Lampje Tourniquet Links Ontgrendelt
LD COM2_TOURN_L  ; TOESTEMMING VRIJG TOURNIKET L
OR M_LAMP_TEST  ; Lamp test d.m.v.Reset zoemer drukknop langer dan 10 seconden ingedrukt te houden
OUT TR0
AND M_STUURSPANNING_IN  ; Merker Stuur Spanning In
OUT Com2_91H14  ; Communicatie Lampje Linkse Tourniquet Ontgrendelt Plc 2 naar Plc 1
LD TR0
OUT 3318.07
; rung 13
LD Com1_91H14  ; Communicatie Lampje Linkse Tourniquet Ontgrendelt Plc 1 naar Plc 2
AND Com2_91H14  ; Communicatie Lampje Linkse Tourniquet Ontgrendelt Plc 2 naar Plc 1
OUT U_91H14  ; TOURNIQUET LINKS ONTGRENDELD
; rung 14: Lampje Tourniquet Rechts Ontgrendelt
LD COM2_TOURN_R  ; TOESTEMMING VRIGAVE TOURNIKET RECHTS
OR M_LAMP_TEST  ; Lamp test d.m.v.Reset zoemer drukknop langer dan 10 seconden ingedrukt te houden
OUT TR0
AND M_STUURSPANNING_IN  ; Merker Stuur Spanning In
OUT Com2_91H16  ; Communicatie Lampje Rechtse Tourniquet Ontgrendelt Plc 2 naar Plc 1
LD TR0
OUT 3318.08
; rung 15
LD Com1_91H16  ; Communicatie Lampje Rechtse Tourniquet Ontgrendelt Plc 1 naar Plc 2
AND Com2_91H16  ; Communicatie Lampje Rechtse Tourniquet Ontgrendelt Plc 2 naar Plc 1
OUT U_91H16  ; TOURNIQUET RECHTS ONTGRENDELD
; rung 16: Lampje Arm & Eiland Omhoog
LD COM2_ARM_OMHOOG  ; PLC 2 ARM OMHOOG
OR M_LAMP_TEST  ; Lamp test d.m.v.Reset zoemer drukknop langer dan 10 seconden ingedrukt te houden
OUT TR0
AND M_STUURSPANNING_IN  ; Merker Stuur Spanning In
OUT Com2_91H18  ; Communicatie Lampje Arm & Eiland Omhoog Plc 2 naar Plc 1
LD TR0
OUT 3320.05
; rung 17
LD Com1_91H18  ; Communicatie Lampje Arm & Eiland Omhoog Plc 1 naar Plc 2
AND Com2_91H18  ; Communicatie Lampje Arm & Eiland Omhoog Plc 2 naar Plc 1
OUT U_91H18  ; ARM (EILAND) OMHOOG

